PROGRAM MAIN
VAR


END_VAR

loopCounter := loopCounter + 1;

PRG_ReadModbusSensorData();			//Temperatur von der Ph-Sonde

(* PRG_HandleUserInputs(); *)

PRG_UpdateMotor();					//Rührmotor

//PRG_UpdateTemperatureControl();		

PRG_UpdatePressureSensor();
PRG_UpdateFlowRateSensor();

Messung1();
//Messung2();

//PRG_UpdatePhControl();
//PRG_UpdateGasSupply();			//Erste Messung nicht nötig
//PRG_UpdateRoomTempRh();			//In Messungen implementiert
//PRG_GasAnalysis();				//Nicht notwendig

END_PROGRAM

(* stored: Version 1.1.0.1, ProductVersion 3.1.4022.12
   POU MAIN: Id {6de127fa-b6f4-4656-b169-9e870eadfc1d}, SpecialFunc None *)
